KUKA KRL data list: openandcheckallclamps.dat

&ACCESS RVO1
&REL 4
&PARAM EDITMASK = *
&PARAM TEMPLATE = C:\KRC\TP\Nutweld\Template\NutWeld_Vorgabe
&PARAM DISKPATH = Program/Utilities
DEFDAT OpenAndCheckAllClamps
;FOLD EXTERNAL DECLARATIONS;%{PE}%MKUKATPBASIS,%CEXT,%VCOMMON,%P
;FOLD BASISTECH EXT;%{PE}%MKUKATPBASIS,%CEXT,%VEXT,%P
EXT  BAS (BAS_COMMAND  :IN,REAL  :IN )
DECL INT SUCCESS
;ENDFOLD (BASISTECH EXT)
;FOLD NutWeld
BOOL NutWeld_TEMPLATE=TRUE
;ENDFOLD (NutWeld)
;FOLD USER EXT;%{E}%MKUKATPUSER,%CEXT,%VEXT,%P
;Make here your modifications

;ENDFOLD (USER EXT)
;ENDFOLD (EXTERNAL DECLARATIONS)
ENDDAT
